// TIA Portal V20 export
// export: Created 2026-09-06T06:46:08.8731269Z, ExportSetting WithDefaults, DisplayName Totally Integrated Automation Portal, DisplayVersion V20, DisplayName TIA Portal Openness, DisplayVersion V20, DisplayName TIA Portal Version Control Interface, DisplayVersion V20, DisplayName STEP 7 Professional, DisplayVersion V20, DisplayName STEP 7 Safety, DisplayVersion V20, DisplayName WinCC Basic/Comfort/Advanced, DisplayVersion V20, DisplayName WinCC Professional, DisplayVersion V20, DisplayName WinCC Unified, DisplayVersion V20
DATA_BLOCK "Valves_DB"   // DB5
{ S7_Optimized_Access := 'TRUE' }
VERSION : 0.1
// stored: AutoNumber true, IsOnlyStoredInLoadMemory false, IsRetainMemResEnabled false, IsWriteProtectedInAS false, MemoryReserve 100
   VAR
      Valve : Array[1..89] of "Valve_IO";
      TotalOpen : Int;
      TotalClosed : Int;
      TotalTransit : Int;
      TotalFault : Int;
      TotalLocal : Int;
      TotalConfigured : Int;
      ErOpen : Int;
      ErClosed : Int;
      ErTransit : Int;
      ErFault : Int;
      ErLocal : Int;
      ErConfigured : Int;
      FwdOpen : Int;
      FwdClosed : Int;
      FwdTransit : Int;
      FwdFault : Int;
      FwdLocal : Int;
      FwdConfigured : Int;
      AftOpen : Int;
      AftClosed : Int;
      AftTransit : Int;
      AftFault : Int;
      AftLocal : Int;
      AftConfigured : Int;
      StateCode : Array[1..89] of Int;
      Stuck : Array[1..89] of Bool;
      Initialized : Array[1..89] of Bool;
      TimeoutOpenAlarm : Array[1..89] of Bool;
      TimeoutCloseAlarm : Array[1..89] of Bool;
      UnexpMove : Array[1..89] of Bool;
      DirFault : Array[1..89] of Bool;
      PosCode : Array[1..89] of Int;
      FaultCode : Array[1..89] of Int;
      CmdPos : Array[1..89] of Int;
      PrevOpenFB : Array[1..89] of Bool;
      PrevClosedFB : Array[1..89] of Bool;
      PosLostTmr : Array[1..89] of TON_TIME;
      DirTmr : Array[1..89] of TON_TIME;
      HwHealthy : Array[1..9] of Bool;
      W_Unhealthy : Array[0..5] of Word;
      W_Conflict : Array[0..5] of Word;
      W_FailOpen : Array[0..5] of Word;
      W_FailClose : Array[0..5] of Word;
      W_LossPos : Array[0..5] of Word;
      W_UnexpMove : Array[0..5] of Word;
      W_Local : Array[0..5] of Word;
      W_DirFault : Array[0..5] of Word;
      HwWord : Word;
      AftPage : Int;
      ErPage : Int;
      FwdPage : Int;
      AftTblState : Array[1..14] of Int;
      ErTblState : Array[1..14] of Int;
      FwdTblState : Array[1..14] of Int;
      AftTblNo : Array[1..14] of Int;
      ErTblNo : Array[1..14] of Int;
      FwdTblNo : Array[1..14] of Int;
      AftTblStateTxt : Array[1..14] of String[14];
      ErTblStateTxt : Array[1..14] of String[14];
      FwdTblStateTxt : Array[1..14] of String[14];
      AftTblTag : Array[1..14] of String[8];
      ErTblTag : Array[1..14] of String[8];
      FwdTblTag : Array[1..14] of String[8];
      CfgPage : Int;
      CfgTblNo : Array[1..16] of Int;
      CfgTblTag : Array[1..16] of String[8];
      CfgTblZone : Array[1..16] of String[12];
      CfgTblConfigured : Array[1..16] of Bool;
      CfgTblState : Array[1..16] of Int;
      CfgTblStateTxt : Array[1..16] of String[14];
      Clock_1Hz : Bool;
      ClockCounter : Int;
      SelIdx : Int;
      SelState : Int;
      SelHealthy : Bool;
      SelLocalMode : Bool;
      SelConfigured : Bool;
      DispCode : Array[1..89] of Int;
      Clock_Flash : Bool;
      HwInitDone : Bool;
   END_VAR
   VAR RETAIN
      ConfiguredRet : Array[1..89] of Bool;
   END_VAR
   VAR
      Clk1Tmr : TON_TIME;
      FlashTmr : TON_TIME;
      WinTmr : TON_TIME;
      PrevAftPage : Int;
      PrevErPage : Int;
      PrevFwdPage : Int;
      PrevCfgPage : Int;
      SelDirFault : Bool;
      SelCmdPos : Int;
      SelPosCode : Int;
      SelFaultCode : Int;
   END_VAR
BEGIN
END_DATA_BLOCK
